// TIA Portal V19 export
TYPE "lexchangetray_typeUnEmn_toRollerDeliver"
// Type: lexchangetray_typeUnEmn_toRollerReq
// Type: lexchangetray_typeUnEmn_toRollerFeedback
// stored: Access Published
   STRUCT
      feedback : "lexchangetray_typeUnEmn_toRollerFeedback";
      req : "lexchangetray_typeUnEmn_toRollerReq";
   END_STRUCT;
END_TYPE
